Fanuc KAREL source: ko00074.KL

PROGRAM KO00074
%STACKSIZE=65535
%PRIORITY=65535
%NOLOCKGROUP
VAR
P1 : XYZWPREXT
P2 : XYZWPREXT
F : BOOLEAN
OUT : XYZWPR
BEGIN
F=TRUE
-- UNSAFE_SOURCE_IR line 11: OUT = MIRROR(P1, convert_xyzwprext_to_position(P2), F)
END KO00074
